Fanuc KAREL source: kb00043.KL

-- PROVISIONAL review KL for V1013-1; original PC SHA256 05ae36f64b47a78c47cb46b77bd40517e3924246e11b3e66b46b1d76962bb2d9
-- Incomplete behavior may be omitted. Consult companion uncertainty JSON. Do not deploy.
PROGRAM KB00043
%NOLOCKGROUP
BEGIN
  -- UNRESOLVED_PC offsets 5-12; opcodes 9D,23
  -- UNRESOLVED_PC offsets 17-26; opcodes 3F,75
  -- UNRESOLVED_PC offsets 31-49; opcodes 27,22,22,2A,31
  -- UNRESOLVED_PC offsets 54-58; opcodes 7F
END KB00043
